PROGRAM MAIN
VAR
	fbAxis: FB_Axis;
	xState: E_MC_State;
	state : BYTE;	
END_VAR

fbAxis.Axis.ReadStatus(); //HMI := gHMI.AxisHMI_1

CASE xState OF
	MCSTATE_Init:		
		fbAxis.Enable(FALSE);		 
		IF fbAxis.Axis.Status.Error THEN
			xState := MCSTATE_Error;
		ELSE	
			xState := MCSTATE_PowerOn;
		END_IF
		
	MCSTATE_PowerOn:
		fbAxis.Enable(TRUE);
		IF fbAxis.power.Done THEN
			xState := MCSTATE_MoveRel;
		END_IF
		
	MCSTATE_Idle:		
		IF gHMI.bMoveRel THEN
			xState:= MCSTATE_MoveRel;
		END_IF
		IF gHMI.bMoveVel THEN
			xState:= MCSTATE_MoveVel;
		END_IF
		IF gHMI.bStop THEN
			xState:= MCSTATE_Stop;
		END_IF
		
	MCSTATE_MoveVel:	
		fbAxis.MoveVel(bExecute := TRUE, Velocity := 100, Direction := MC_Positive_Direction, 						
						acceleration := 1000, Deceleration := 1500, Jerk:= 0);	
		IF fbAxis.moveVels.Active THEN
			fbAxis.MoveVel(bExecute := FALSE, Velocity := 100, Direction := MC_Positive_Direction, 
						acceleration := 1000, Deceleration := 1500, Jerk:= 0);	
		END_IF
		IF gHMI.bStop THEN
			xState:= MCSTATE_Stop;
		END_IF
		
	MCSTATE_Stop:		
		fbAxis.Stop(bExecute := TRUE, Deceleration := 1500, Jerk:= 0);
		IF fbAxis.stops.Done  THEN
			fbAxis.Stop(bExecute := FALSE, Deceleration := 1500, Jerk:= 0);			
			xState := MCSTATE_Idle;
		END_IF
				
	MCSTATE_MoveRel:
		fbAxis.MoveRel(bExecute:=TRUE,relAngle:=100);		 
		IF fbAxis.moveRels.Done THEN
			fbAxis.MoveRel(bExecute:=FALSE,relAngle:=100);	
			xState := MCSTATE_Idle;
		END_IF
END_CASE

END_PROGRAM

(* stored: Version 1.1.0.1, ProductVersion 3.1.4024.0
   POU MAIN: Id {9e1c3995-83c8-4182-bd18-563ee53d3d94}, SpecialFunc None *)
